// TIA Portal V19 export
FUNCTION "Loop1_CALL" : Void   // FC165, LAD
TITLE = LOOP 1 - ENTRY = COIL HANDLING ZONE / EXIT = POST-PUNCHING ZONE
// stored: SetENOAutomatically false
   VAR_TEMP
      Dummy : Bool;
   END_VAR
   VAR_TEMP   // added for the SCL form of the ladder/FBD networks
      _w1 : Bool;
   END_VAR
BEGIN

REGION Network 1: Data In
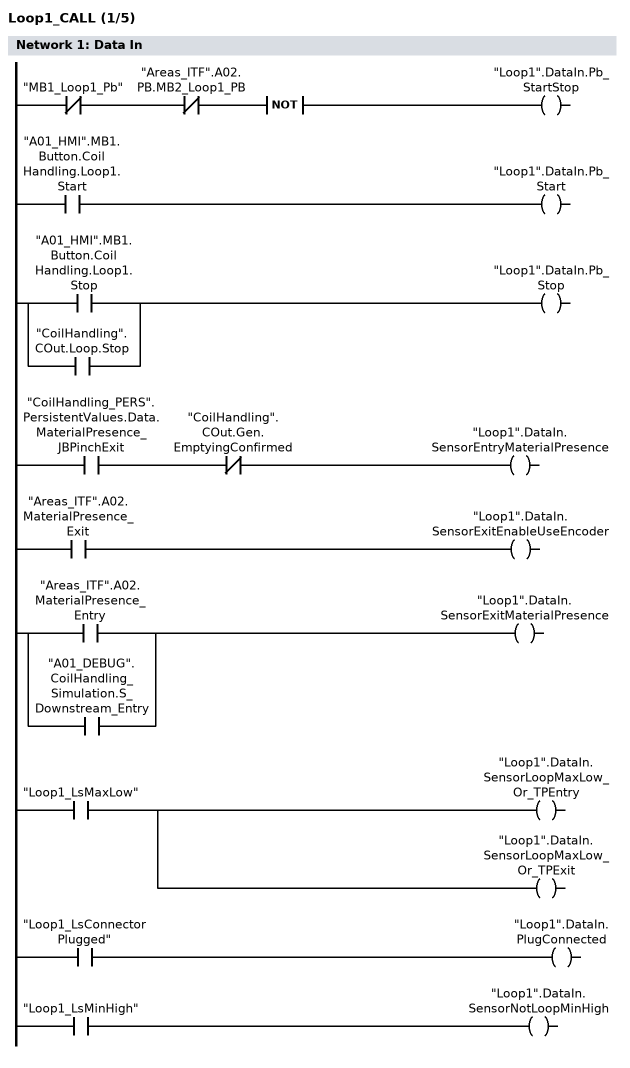
   RUNG wire#powerrail
      I_Contact( "MB1_Loop1_Pb" )
      I_Contact( "Areas_ITF".A02.PB.MB2_Loop1_PB )
      Not()
      Coil( "Loop1".DataIn.Pb_StartStop )
   END_RUNG
   RUNG wire#powerrail
      Contact( "A01_HMI".MB1.Button.CoilHandling.Loop1.Start )
      Coil( "Loop1".DataIn.Pb_Start )
   END_RUNG
   RUNG wire#powerrail
      Contact( "A01_HMI".MB1.Button.CoilHandling.Loop1.Stop )
      wire#w1
      Coil( "Loop1".DataIn.Pb_Stop )
   END_RUNG
   RUNG wire#powerrail
      Contact( "CoilHandling".COut.Loop.Stop )
   END_RUNG wire#w1
   RUNG wire#powerrail
      Contact( "CoilHandling_PERS".PersistentValues.Data.MaterialPresence_JBPinchExit )
      I_Contact( "CoilHandling".COut.Gen.EmptyingConfirmed )
      Coil( "Loop1".DataIn.SensorEntryMaterialPresence )
   END_RUNG
   RUNG wire#powerrail
      Contact( "Areas_ITF".A02.MaterialPresence_Exit )
      Coil( "Loop1".DataIn.SensorExitEnableUseEncoder )
   END_RUNG
   RUNG wire#powerrail
      Contact( "Areas_ITF".A02.MaterialPresence_Entry )
      wire#w2
      Coil( "Loop1".DataIn.SensorExitMaterialPresence )
   END_RUNG
   RUNG wire#powerrail
      Contact( "A01_DEBUG".CoilHandling_Simulation.S_Downstream_Entry )
   END_RUNG wire#w2
   RUNG wire#powerrail
      Contact( "Loop1_LsMaxLow" )
      wire#w3
      Coil( "Loop1".DataIn.SensorLoopMaxLow_Or_TPEntry )
   END_RUNG
   RUNG wire#w3
      Coil( "Loop1".DataIn.SensorLoopMaxLow_Or_TPExit )
   END_RUNG
   RUNG wire#powerrail
      Contact( "Loop1_LsConnectorPlugged" )
      Coil( "Loop1".DataIn.PlugConnected )
   END_RUNG
   RUNG wire#powerrail
      Contact( "Loop1_LsMinHigh" )
      Coil( "Loop1".DataIn.SensorNotLoopMinHigh )
   END_RUNG
   // the same network as SCL:
   "Loop1".DataIn.Pb_StartStop := NOT (NOT "MB1_Loop1_Pb" AND NOT "Areas_ITF".A02.PB.MB2_Loop1_PB);
   "Loop1".DataIn.Pb_Start := "A01_HMI".MB1.Button.CoilHandling.Loop1.Start;
   "Loop1".DataIn.Pb_Stop := "A01_HMI".MB1.Button.CoilHandling.Loop1.Stop OR "CoilHandling".COut.Loop.Stop;
   "Loop1".DataIn.SensorEntryMaterialPresence := "CoilHandling_PERS".PersistentValues.Data.MaterialPresence_JBPinchExit AND NOT "CoilHandling".COut.Gen.EmptyingConfirmed;
   "Loop1".DataIn.SensorExitEnableUseEncoder := "Areas_ITF".A02.MaterialPresence_Exit;
   "Loop1".DataIn.SensorExitMaterialPresence := "Areas_ITF".A02.MaterialPresence_Entry OR "A01_DEBUG".CoilHandling_Simulation.S_Downstream_Entry;
   "Loop1".DataIn.SensorLoopMaxLow_Or_TPEntry := "Loop1_LsMaxLow";
   "Loop1".DataIn.SensorLoopMaxLow_Or_TPExit := "Loop1_LsMaxLow";
   "Loop1".DataIn.PlugConnected := "Loop1_LsConnectorPlugged";
   "Loop1".DataIn.SensorNotLoopMinHigh := "Loop1_LsMinHigh";
END_REGION

REGION Network 2: >
END_REGION

REGION Network 3: Coordination In
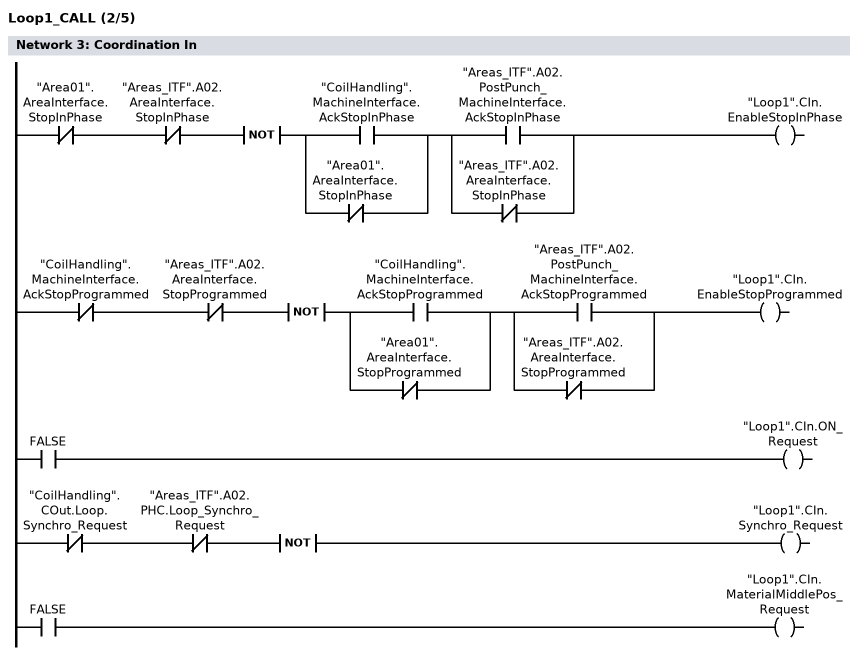
   RUNG wire#powerrail
      I_Contact( "Area01".AreaInterface.StopInPhase )
      I_Contact( "Areas_ITF".A02.AreaInterface.StopInPhase )
      Not()
      wire#w1
      Contact( "CoilHandling".MachineInterface.AckStopInPhase )
      wire#w2
      Contact( "Areas_ITF".A02.PostPunch_MachineInterface.AckStopInPhase )
      wire#w3
      Coil( "Loop1".CIn.EnableStopInPhase )
   END_RUNG
   RUNG wire#w1
      I_Contact( "Area01".AreaInterface.StopInPhase )
   END_RUNG wire#w2
   RUNG wire#w2
      I_Contact( "Areas_ITF".A02.AreaInterface.StopInPhase )
   END_RUNG wire#w3
   RUNG wire#powerrail
      I_Contact( "CoilHandling".MachineInterface.AckStopProgrammed )
      I_Contact( "Areas_ITF".A02.AreaInterface.StopProgrammed )
      Not()
      wire#w4
      Contact( "CoilHandling".MachineInterface.AckStopProgrammed )
      wire#w5
      Contact( "Areas_ITF".A02.PostPunch_MachineInterface.AckStopProgrammed )
      wire#w6
      Coil( "Loop1".CIn.EnableStopProgrammed )
   END_RUNG
   RUNG wire#w4
      I_Contact( "Area01".AreaInterface.StopProgrammed )
   END_RUNG wire#w5
   RUNG wire#w5
      I_Contact( "Areas_ITF".A02.AreaInterface.StopProgrammed )
   END_RUNG wire#w6
   RUNG wire#powerrail
      Contact( FALSE )
      Coil( "Loop1".CIn.ON_Request )
   END_RUNG
   RUNG wire#powerrail
      I_Contact( "CoilHandling".COut.Loop.Synchro_Request )
      I_Contact( "Areas_ITF".A02.PHC.Loop_Synchro_Request )
      Not()
      Coil( "Loop1".CIn.Synchro_Request )
   END_RUNG
   RUNG wire#powerrail
      Contact( FALSE )
      Coil( "Loop1".CIn.MaterialMiddlePos_Request )
   END_RUNG
   // the same network as SCL:
   "Loop1".CIn.EnableStopInPhase := NOT (NOT "Area01".AreaInterface.StopInPhase AND NOT "Areas_ITF".A02.AreaInterface.StopInPhase) AND ("CoilHandling".MachineInterface.AckStopInPhase OR NOT "Area01".AreaInterface.StopInPhase) AND ("Areas_ITF".A02.PostPunch_MachineInterface.AckStopInPhase OR NOT "Areas_ITF".A02.AreaInterface.StopInPhase);
   "Loop1".CIn.EnableStopProgrammed := NOT (NOT "CoilHandling".MachineInterface.AckStopProgrammed AND NOT "Areas_ITF".A02.AreaInterface.StopProgrammed) AND ("CoilHandling".MachineInterface.AckStopProgrammed OR NOT "Area01".AreaInterface.StopProgrammed) AND ("Areas_ITF".A02.PostPunch_MachineInterface.AckStopProgrammed OR NOT "Areas_ITF".A02.AreaInterface.StopProgrammed);
   "Loop1".CIn.ON_Request := FALSE;
   "Loop1".CIn.Synchro_Request := NOT (NOT "CoilHandling".COut.Loop.Synchro_Request AND NOT "Areas_ITF".A02.PHC.Loop_Synchro_Request);
   "Loop1".CIn.MaterialMiddlePos_Request := FALSE;
END_REGION

REGION Network 4: Coordination In - Entry
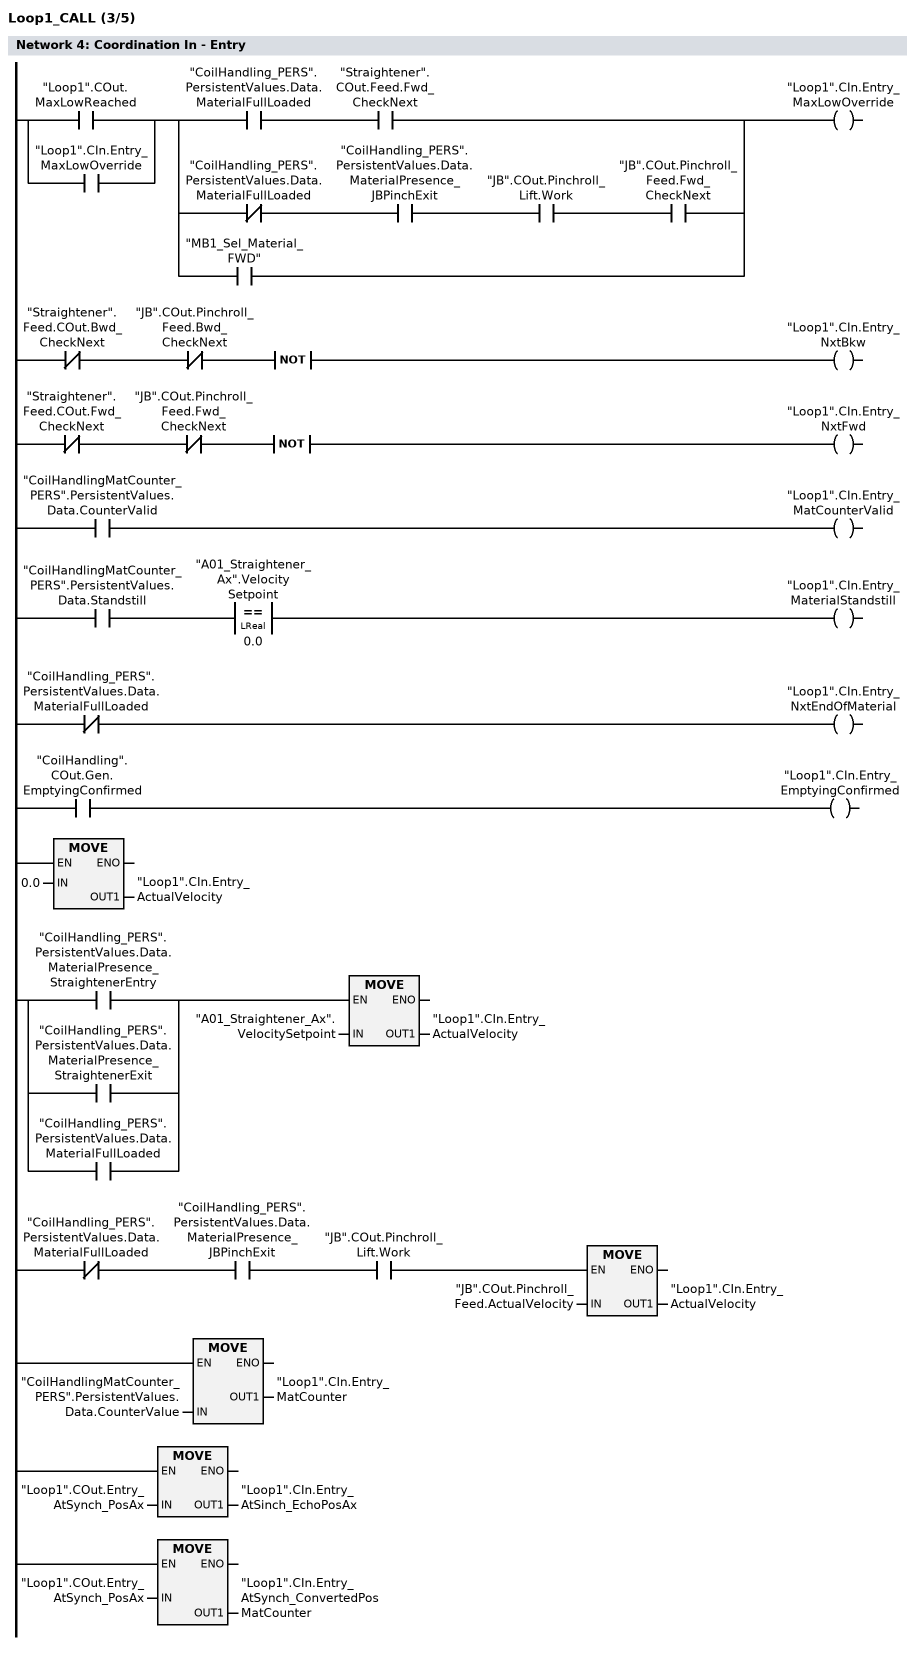
   RUNG wire#powerrail
      Contact( "Loop1".COut.MaxLowReached )
      wire#w1
      Contact( "CoilHandling_PERS".PersistentValues.Data.MaterialFullLoaded )
      Contact( "Straightener".COut.Feed.Fwd_CheckNext )
      wire#w2
      Coil( "Loop1".CIn.Entry_MaxLowOverride )
   END_RUNG
   RUNG wire#powerrail
      Contact( "Loop1".CIn.Entry_MaxLowOverride )
   END_RUNG wire#w1
   RUNG wire#w1
      I_Contact( "CoilHandling_PERS".PersistentValues.Data.MaterialFullLoaded )
      Contact( "CoilHandling_PERS".PersistentValues.Data.MaterialPresence_JBPinchExit )
      Contact( "JB".COut.Pinchroll_Lift.Work )
      Contact( "JB".COut.Pinchroll_Feed.Fwd_CheckNext )
   END_RUNG wire#w2
   RUNG wire#w1
      Contact( "MB1_Sel_Material_FWD" )
   END_RUNG wire#w2
   RUNG wire#powerrail
      I_Contact( "Straightener".Feed.COut.Bwd_CheckNext )
      I_Contact( "JB".COut.Pinchroll_Feed.Bwd_CheckNext )
      Not()
      Coil( "Loop1".CIn.Entry_NxtBkw )
   END_RUNG
   RUNG wire#powerrail
      I_Contact( "Straightener".Feed.COut.Fwd_CheckNext )
      I_Contact( "JB".COut.Pinchroll_Feed.Fwd_CheckNext )
      Not()
      Coil( "Loop1".CIn.Entry_NxtFwd )
   END_RUNG
   RUNG wire#powerrail
      Contact( "CoilHandlingMatCounter_PERS".PersistentValues.Data.CounterValid )
      Coil( "Loop1".CIn.Entry_MatCounterValid )
   END_RUNG
   RUNG wire#powerrail
      Contact( "CoilHandlingMatCounter_PERS".PersistentValues.Data.Standstill )
      { S7_Templates := "SrcType := LReal" } EQ_Contact(in1 := "A01_Straightener_Ax".VelocitySetpoint, in2 := 0.0)
      Coil( "Loop1".CIn.Entry_MaterialStandstill )
   END_RUNG
   RUNG wire#powerrail
      I_Contact( "CoilHandling_PERS".PersistentValues.Data.MaterialFullLoaded )
      Coil( "Loop1".CIn.Entry_NxtEndOfMaterial )
   END_RUNG
   RUNG wire#powerrail
      Contact( "CoilHandling".COut.Gen.EmptyingConfirmed )
      Coil( "Loop1".CIn.Entry_EmptyingConfirmed )
   END_RUNG
   RUNG wire#powerrail
      { S7_GenerateENO := "TRUE" } Move(in := 0.0, out1 => "Loop1".CIn.Entry_ActualVelocity)
   END_RUNG
   RUNG wire#powerrail
      Contact( "CoilHandling_PERS".PersistentValues.Data.MaterialPresence_StraightenerEntry )
      wire#w3
      Move(in := "A01_Straightener_Ax".VelocitySetpoint, out1 => "Loop1".CIn.Entry_ActualVelocity)
   END_RUNG
   RUNG wire#powerrail
      Contact( "CoilHandling_PERS".PersistentValues.Data.MaterialPresence_StraightenerExit )
   END_RUNG wire#w3
   RUNG wire#powerrail
      Contact( "CoilHandling_PERS".PersistentValues.Data.MaterialFullLoaded )
   END_RUNG wire#w3
   RUNG wire#powerrail
      I_Contact( "CoilHandling_PERS".PersistentValues.Data.MaterialFullLoaded )
      Contact( "CoilHandling_PERS".PersistentValues.Data.MaterialPresence_JBPinchExit )
      Contact( "JB".COut.Pinchroll_Lift.Work )
      Move(in := "JB".COut.Pinchroll_Feed.ActualVelocity, out1 => "Loop1".CIn.Entry_ActualVelocity)
   END_RUNG
   RUNG wire#powerrail
      Move(in := "CoilHandlingMatCounter_PERS".PersistentValues.Data.CounterValue, out1 => "Loop1".CIn.Entry_MatCounter)
   END_RUNG
   RUNG wire#powerrail
      Move(in := "Loop1".COut.Entry_AtSynch_PosAx, out1 => "Loop1".CIn.Entry_AtSinch_EchoPosAx)
   END_RUNG
   RUNG wire#powerrail
      Move(in := "Loop1".COut.Entry_AtSynch_PosAx, out1 => "Loop1".CIn.Entry_AtSynch_ConvertedPosMatCounter)
   END_RUNG
   // the same network as SCL:
   "Loop1".CIn.Entry_MaxLowOverride := ("Loop1".COut.MaxLowReached OR "Loop1".CIn.Entry_MaxLowOverride) AND (("CoilHandling_PERS".PersistentValues.Data.MaterialFullLoaded AND "Straightener".COut.Feed.Fwd_CheckNext) OR (NOT "CoilHandling_PERS".PersistentValues.Data.MaterialFullLoaded AND "CoilHandling_PERS".PersistentValues.Data.MaterialPresence_JBPinchExit AND "JB".COut.Pinchroll_Lift.Work AND "JB".COut.Pinchroll_Feed.Fwd_CheckNext) OR "MB1_Sel_Material_FWD");
   "Loop1".CIn.Entry_NxtBkw := NOT (NOT "Straightener".Feed.COut.Bwd_CheckNext AND NOT "JB".COut.Pinchroll_Feed.Bwd_CheckNext);
   "Loop1".CIn.Entry_NxtFwd := NOT (NOT "Straightener".Feed.COut.Fwd_CheckNext AND NOT "JB".COut.Pinchroll_Feed.Fwd_CheckNext);
   "Loop1".CIn.Entry_MatCounterValid := "CoilHandlingMatCounter_PERS".PersistentValues.Data.CounterValid;
   "Loop1".CIn.Entry_MaterialStandstill := "CoilHandlingMatCounter_PERS".PersistentValues.Data.Standstill AND ("A01_Straightener_Ax".VelocitySetpoint = 0.0);
   "Loop1".CIn.Entry_NxtEndOfMaterial := NOT "CoilHandling_PERS".PersistentValues.Data.MaterialFullLoaded;
   "Loop1".CIn.Entry_EmptyingConfirmed := "CoilHandling".COut.Gen.EmptyingConfirmed;
   "Loop1".CIn.Entry_ActualVelocity := 0.0;
   IF "CoilHandling_PERS".PersistentValues.Data.MaterialPresence_StraightenerEntry OR "CoilHandling_PERS".PersistentValues.Data.MaterialPresence_StraightenerExit OR "CoilHandling_PERS".PersistentValues.Data.MaterialFullLoaded THEN
       "Loop1".CIn.Entry_ActualVelocity := "A01_Straightener_Ax".VelocitySetpoint;
   END_IF;
   IF NOT "CoilHandling_PERS".PersistentValues.Data.MaterialFullLoaded AND "CoilHandling_PERS".PersistentValues.Data.MaterialPresence_JBPinchExit AND "JB".COut.Pinchroll_Lift.Work THEN
       "Loop1".CIn.Entry_ActualVelocity := "JB".COut.Pinchroll_Feed.ActualVelocity;
   END_IF;
   "Loop1".CIn.Entry_MatCounter := "CoilHandlingMatCounter_PERS".PersistentValues.Data.CounterValue;
   "Loop1".CIn.Entry_AtSinch_EchoPosAx := "Loop1".COut.Entry_AtSynch_PosAx;
   "Loop1".CIn.Entry_AtSynch_ConvertedPosMatCounter := "Loop1".COut.Entry_AtSynch_PosAx;
END_REGION

REGION Network 5: Coordination In - Exit
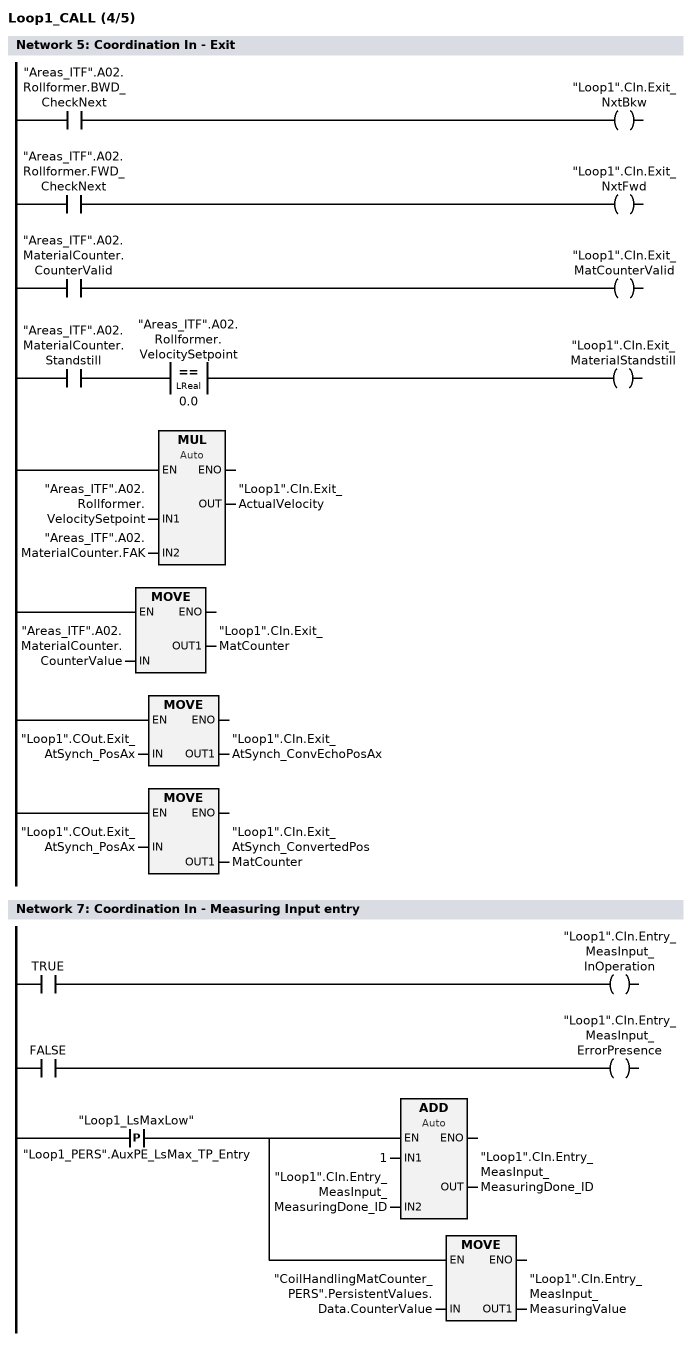
   RUNG wire#powerrail
      Contact( "Areas_ITF".A02.Rollformer.BWD_CheckNext )
      Coil( "Loop1".CIn.Exit_NxtBkw )
   END_RUNG
   RUNG wire#powerrail
      Contact( "Areas_ITF".A02.Rollformer.FWD_CheckNext )
      Coil( "Loop1".CIn.Exit_NxtFwd )
   END_RUNG
   RUNG wire#powerrail
      Contact( "Areas_ITF".A02.MaterialCounter.CounterValid )
      Coil( "Loop1".CIn.Exit_MatCounterValid )
   END_RUNG
   RUNG wire#powerrail
      Contact( "Areas_ITF".A02.MaterialCounter.Standstill )
      { S7_Templates := "SrcType := LReal" } EQ_Contact(in1 := "Areas_ITF".A02.Rollformer.VelocitySetpoint, in2 := 0.0)
      Coil( "Loop1".CIn.Exit_MaterialStandstill )
   END_RUNG
   RUNG wire#powerrail
      { S7_GenerateENO := "TRUE" } Mul(in1 := "Areas_ITF".A02.Rollformer.VelocitySetpoint, in2 := "Areas_ITF".A02.MaterialCounter.FAK, out => "Loop1".CIn.Exit_ActualVelocity)
   END_RUNG
   RUNG wire#powerrail
      Move(in := "Areas_ITF".A02.MaterialCounter.CounterValue, out1 => "Loop1".CIn.Exit_MatCounter)
   END_RUNG
   RUNG wire#powerrail
      Move(in := "Loop1".COut.Exit_AtSynch_PosAx, out1 => "Loop1".CIn.Exit_AtSynch_ConvEchoPosAx)
   END_RUNG
   RUNG wire#powerrail
      Move(in := "Loop1".COut.Exit_AtSynch_PosAx, out1 => "Loop1".CIn.Exit_AtSynch_ConvertedPosMatCounter)
   END_RUNG
   // the same network as SCL:
   "Loop1".CIn.Exit_NxtBkw := "Areas_ITF".A02.Rollformer.BWD_CheckNext;
   "Loop1".CIn.Exit_NxtFwd := "Areas_ITF".A02.Rollformer.FWD_CheckNext;
   "Loop1".CIn.Exit_MatCounterValid := "Areas_ITF".A02.MaterialCounter.CounterValid;
   "Loop1".CIn.Exit_MaterialStandstill := "Areas_ITF".A02.MaterialCounter.Standstill AND ("Areas_ITF".A02.Rollformer.VelocitySetpoint = 0.0);
   "Loop1".CIn.Exit_ActualVelocity := "Areas_ITF".A02.Rollformer.VelocitySetpoint * "Areas_ITF".A02.MaterialCounter.FAK;
   "Loop1".CIn.Exit_MatCounter := "Areas_ITF".A02.MaterialCounter.CounterValue;
   "Loop1".CIn.Exit_AtSynch_ConvEchoPosAx := "Loop1".COut.Exit_AtSynch_PosAx;
   "Loop1".CIn.Exit_AtSynch_ConvertedPosMatCounter := "Loop1".COut.Exit_AtSynch_PosAx;
END_REGION

REGION Network 6: >
END_REGION

REGION Network 7: Coordination In - Measuring Input entry
   RUNG wire#powerrail
      Contact( TRUE )
      Coil( "Loop1".CIn.Entry_MeasInput_InOperation )
   END_RUNG
   RUNG wire#powerrail
      Contact( FALSE )
      Coil( "Loop1".CIn.Entry_MeasInput_ErrorPresence )
   END_RUNG
   RUNG wire#powerrail
      P_Contact(operand := "Loop1_LsMaxLow", bit := "Loop1_PERS".AuxPE_LsMax_TP_Entry)
      wire#w1
      Add(in1 := 1, in2 := "Loop1".CIn.Entry_MeasInput_MeasuringDone_ID, out => "Loop1".CIn.Entry_MeasInput_MeasuringDone_ID)
   END_RUNG
   RUNG wire#w1
      Move(in := "CoilHandlingMatCounter_PERS".PersistentValues.Data.CounterValue, out1 => "Loop1".CIn.Entry_MeasInput_MeasuringValue)
   END_RUNG
   // the same network as SCL:
   "Loop1".CIn.Entry_MeasInput_InOperation := TRUE;
   "Loop1".CIn.Entry_MeasInput_ErrorPresence := FALSE;
   #_w1 := "Loop1_LsMaxLow" AND NOT "Loop1_PERS".AuxPE_LsMax_TP_Entry;   // rising edge of "Loop1_LsMaxLow"
   "Loop1_PERS".AuxPE_LsMax_TP_Entry := "Loop1_LsMaxLow";
   IF #_w1 THEN
       "Loop1".CIn.Entry_MeasInput_MeasuringDone_ID := 1 + "Loop1".CIn.Entry_MeasInput_MeasuringDone_ID;
       "Loop1".CIn.Entry_MeasInput_MeasuringValue := "CoilHandlingMatCounter_PERS".PersistentValues.Data.CounterValue;
   END_IF;
END_REGION

REGION Network 8: Coordination In - Measuring Input exit
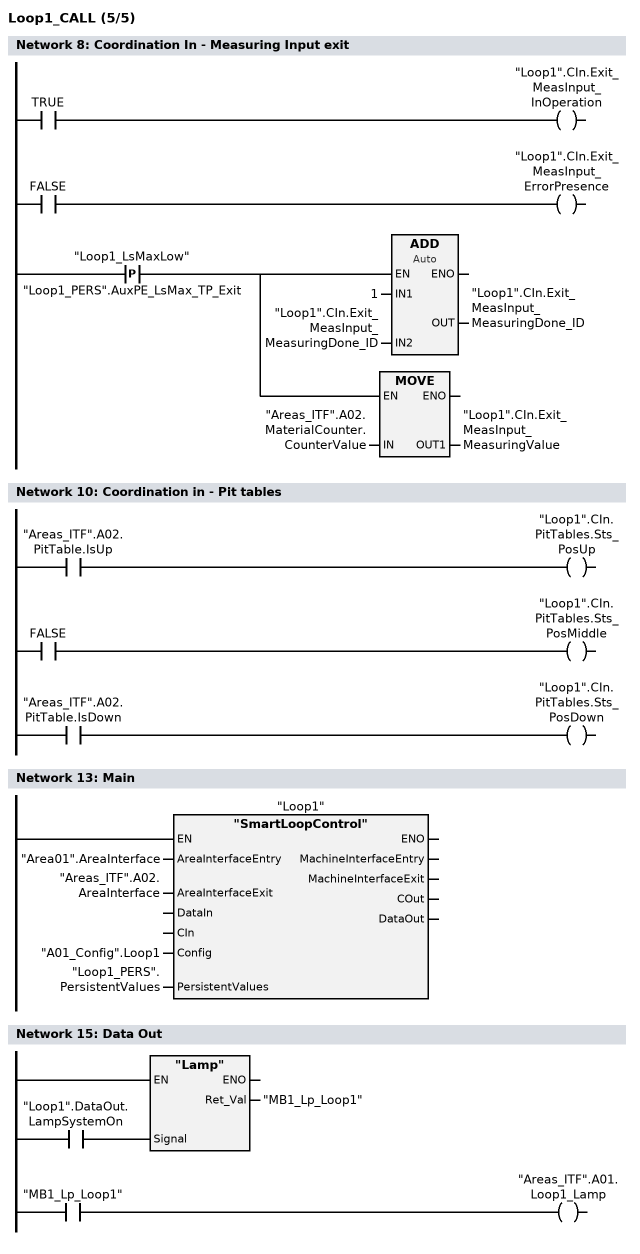
   RUNG wire#powerrail
      Contact( TRUE )
      Coil( "Loop1".CIn.Exit_MeasInput_InOperation )
   END_RUNG
   RUNG wire#powerrail
      Contact( FALSE )
      Coil( "Loop1".CIn.Exit_MeasInput_ErrorPresence )
   END_RUNG
   RUNG wire#powerrail
      P_Contact(operand := "Loop1_LsMaxLow", bit := "Loop1_PERS".AuxPE_LsMax_TP_Exit)
      wire#w1
      Add(in1 := 1, in2 := "Loop1".CIn.Exit_MeasInput_MeasuringDone_ID, out => "Loop1".CIn.Exit_MeasInput_MeasuringDone_ID)
   END_RUNG
   RUNG wire#w1
      Move(in := "Areas_ITF".A02.MaterialCounter.CounterValue, out1 => "Loop1".CIn.Exit_MeasInput_MeasuringValue)
   END_RUNG
   // the same network as SCL:
   "Loop1".CIn.Exit_MeasInput_InOperation := TRUE;
   "Loop1".CIn.Exit_MeasInput_ErrorPresence := FALSE;
   #_w1 := "Loop1_LsMaxLow" AND NOT "Loop1_PERS".AuxPE_LsMax_TP_Exit;   // rising edge of "Loop1_LsMaxLow"
   "Loop1_PERS".AuxPE_LsMax_TP_Exit := "Loop1_LsMaxLow";
   IF #_w1 THEN
       "Loop1".CIn.Exit_MeasInput_MeasuringDone_ID := 1 + "Loop1".CIn.Exit_MeasInput_MeasuringDone_ID;
       "Loop1".CIn.Exit_MeasInput_MeasuringValue := "Areas_ITF".A02.MaterialCounter.CounterValue;
   END_IF;
END_REGION

REGION Network 9: >
END_REGION

REGION Network 10: Coordination in - Pit tables
   RUNG wire#powerrail
      Contact( "Areas_ITF".A02.PitTable.IsUp )
      Coil( "Loop1".CIn.PitTables.Sts_PosUp )
   END_RUNG
   RUNG wire#powerrail
      Contact( FALSE )
      Coil( "Loop1".CIn.PitTables.Sts_PosMiddle )
   END_RUNG
   RUNG wire#powerrail
      Contact( "Areas_ITF".A02.PitTable.IsDown )
      Coil( "Loop1".CIn.PitTables.Sts_PosDown )
   END_RUNG
   // the same network as SCL:
   "Loop1".CIn.PitTables.Sts_PosUp := "Areas_ITF".A02.PitTable.IsUp;
   "Loop1".CIn.PitTables.Sts_PosMiddle := FALSE;
   "Loop1".CIn.PitTables.Sts_PosDown := "Areas_ITF".A02.PitTable.IsDown;
END_REGION

REGION Network 11: >
END_REGION

REGION Network 12: >
END_REGION

REGION Network 13: Main
   RUNG wire#powerrail
      "Loop1"(AreaInterfaceEntry := "Area01".AreaInterface, AreaInterfaceExit := "Areas_ITF".A02.AreaInterface, DataIn :=, CIn :=, Config := "A01_Config".Loop1, PersistentValues := "Loop1_PERS".PersistentValues, MachineInterfaceEntry =>, MachineInterfaceExit =>, COut =>, DataOut =>)
   END_RUNG
   // the same network as SCL:
   "Loop1"(AreaInterfaceEntry := "Area01".AreaInterface,   // "SmartLoopControl"
           AreaInterfaceExit := "Areas_ITF".A02.AreaInterface,
           Config := "A01_Config".Loop1,
           PersistentValues := "Loop1_PERS".PersistentValues);
END_REGION

REGION Network 14: >
END_REGION

REGION Network 15: Data Out
   RUNG wire#powerrail
      "Lamp"(Signal := wire#w1, Ret_Val => "MB1_Lp_Loop1")
   END_RUNG
   RUNG wire#powerrail
      Contact( "Loop1".DataOut.LampSystemOn )
   END_RUNG wire#w1
   RUNG wire#powerrail
      Contact( "MB1_Lp_Loop1" )
      Coil( "Areas_ITF".A01.Loop1_Lamp )
   END_RUNG
   // the same network as SCL:
   "MB1_Lp_Loop1" := "Lamp"(Signal := "Loop1".DataOut.LampSystemOn);
   "Areas_ITF".A01.Loop1_Lamp := "MB1_Lp_Loop1";
END_REGION

REGION Network 16: >
END_REGION

REGION Network 17: >
END_REGION

REGION Network 18: >
END_REGION
END_FUNCTION
